{attribute 'qualified_only'}
VAR_GLOBAL CONSTANT
	nSAFETY_OUTPUTS: UINT := 8; //do these break with a 0 value?
	nSAFETY_DEVICES: UINT := 1;
	nSAFETY_OUTPUT_GROUPS: UINT := 3;
END_VAR

(* stored: Version 1.1.0.1, ProductVersion 3.1.4024.11
   GVL GVL_Safety: Id {77e096dc-056c-4248-bab4-5cc16df9938e} *)
